TYPE GearInDyn_CMD_typ :
STRUCT
	StartSlave : BOOL ;
	DisengageSlave : BOOL ;
END_STRUCT
END_TYPE

(* stored: Version 1.1.0.1, ProductVersion 3.1.4024.3
   DUT GearInDyn_CMD_typ: Id {d37e81d7-8644-0e0c-3b13-b58db0515353} *)
